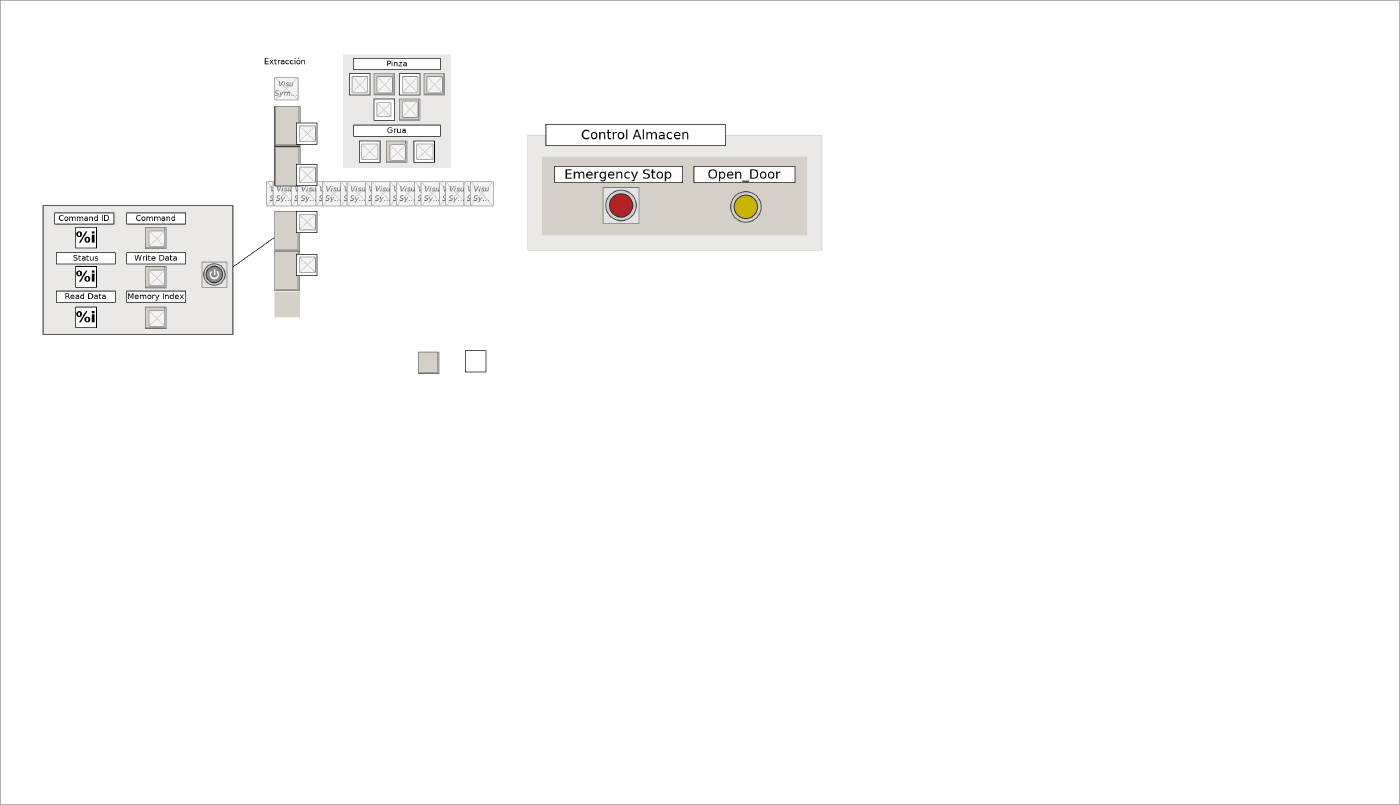
VISUALIZATION Almacen_Manual  // 1930x1110
    Rectangle (369,356 55x35), angle 90
    Group (367,250 330x48)
        Group (0,0 126x48)
            Group (0,0 92x48)
                Group (0,0 58x48)
                    Rectangle (8,5 24x23)
                    Image (0,0 32x34), image: VisuSymbols.Symbols.ArrowForward
                    Image (9,0 32x34), angle 90, image: VisuSymbols.Symbols.ArrowDown
                Group (34,0 58x48)
                    Rectangle (8,5 24x23)
                    Image (0,0 32x34), image: VisuSymbols.Symbols.ArrowForward
                    Image (9,0 32x34), angle 90, image: VisuSymbols.Symbols.ArrowDown
            Group (68,0 58x48)
                Rectangle (8,5 24x23)
                Image (0,0 32x34), image: VisuSymbols.Symbols.ArrowForward
                Image (9,0 32x34), angle 90, image: VisuSymbols.Symbols.ArrowDown
        Group (102,0 126x48)
            Group (0,0 92x48)
                Group (0,0 58x48)
                    Rectangle (8,5 24x23)
                    Image (0,0 32x34), image: VisuSymbols.Symbols.ArrowForward
                    Image (9,0 32x34), angle 90, image: VisuSymbols.Symbols.ArrowDown
                Group (34,0 58x48)
                    Rectangle (8,5 24x23)
                    Image (0,0 32x34), image: VisuSymbols.Symbols.ArrowForward
                    Image (9,0 32x34), angle 90, image: VisuSymbols.Symbols.ArrowDown
            Group (68,0 58x48)
                Rectangle (8,5 24x23)
                Image (0,0 32x34), image: VisuSymbols.Symbols.ArrowForward
                Image (9,0 32x34), angle 90, image: VisuSymbols.Symbols.ArrowDown
        Group (204,0 126x48)
            Group (0,0 92x48)
                Group (0,0 58x48)
                    Rectangle (8,5 24x23)
                    Image (0,0 32x34), image: VisuSymbols.Symbols.ArrowForward
                    Image (9,0 32x34), angle 90, image: VisuSymbols.Symbols.ArrowDown
                Group (34,0 58x48)
                    Rectangle (8,5 24x23)
                    Image (0,0 32x34), image: VisuSymbols.Symbols.ArrowForward
                    Image (9,0 32x34), angle 90, image: VisuSymbols.Symbols.ArrowDown
            Group (68,0 58x48)
                Rectangle (8,5 24x23)
                Image (0,0 32x34), image: VisuSymbols.Symbols.ArrowForward
                Image (9,0 32x34), angle 90, image: VisuSymbols.Symbols.ArrowDown
    InvisibleInput (355,103 77x35)
    Image (378,106 33x32), image: VisuSymbols.Symbols.ForwardStandard
    Rectangle (347,76 92x18), "Extracción"
    Rectangle (379,402 35x35), angle 90
    Rectangle (369,301 55x35), angle 90
    Rectangle (369,211 55x35), angle 90
    Rectangle (369,156 55x35), angle 90
    InvisibleInput (1163,198 18x136)
    Line (377,328) (318,370)
    InvisibleInput (262,497 18x41)
    Rectangle (1771,538 159x406), angle 90
    Rectangle (752,171 248x30), "Control Almacen"
    Rectangle (1780,528 108x365), angle 90
    PushSwitch (831,258 50x50), variable: GVL.Emergency_Stop_9, behaviour: TOGGLE, style: Switch-PushSwitch-Red
    Rectangle (764,229 177x23), "Emergency Stop"
    Lamp1 (1003,260 50x50), variable: NOT GVL.Safety_Door_13 OR NOT GVL.Safety_Door_14 OR NOT GVL.Safety_Door_15, style: Lamp-Lamp1-Yellow
    Rectangle (956,229 140x23), "Open_Door"
    Rectangle (1198,848 178x262), angle 90
    Rectangle (104,313 29x29), "%i", text variable: GVL.RFID_Reader_1_Command_ID
        p4168582468: GVL.RFID_Reader_1_Command_ID
    Rectangle (75,293 82x16), "Command ID"
    Rectangle (77,348 82x16), "Status"
    Rectangle (77,401 82x16), "Read Data"
    Rectangle (104,367 29x29), "%i", text variable: GVL.RFID_Reader_1_Status
        p4168582468: GVL.RFID_Reader_1_Status
    Rectangle (104,423 29x29), "%i", text variable: GVL.RFID_Reader_1_Read_Data
        p4168582468: GVL.RFID_Reader_1_Read_Data
    PowerSwitch (278,361 35x35), variable: GVL.RFID_Reader_1_Ejecute_Comm, behaviour: TOGGLE, style: Switch-PowerSwitch-Gray
    Button (378,346 35x55), colour toggle: GVL.Roller_Conveyor_2m_8, pressed state: GVL.Roller_Conveyor_2m_8
        OnMouseClick: toggle GVL.Roller_Conveyor_2m_8
    Button (378,291 35x55), colour toggle: GVL.Loading_Conveyor_1, pressed state: GVL.Loading_Conveyor_1
        OnMouseClick: toggle GVL.Loading_Conveyor_1
    Group (408,291 29x30), colour toggle: GVL.Retroreflective_Sensor_1
        RoundedRectangle (0,0 29x30), colour toggle: GVL.Diffuse_Sensor_4
        Image (4,4 23x22), image: VisuSymbols.Symbols.RSS1
    Group (408,350 29x30), colour toggle: GVL.Diffuse_Sensor_43
        RoundedRectangle (0,0 29x30), colour toggle: GVL.Diffuse_Sensor_4
        Image (4,4 23x22), image: VisuSymbols.Symbols.RSS1
    Button (379,202 35x55), colour toggle: GVL.Loading_Conveyor_2, pressed state: GVL.Loading_Conveyor_2
        OnMouseClick: toggle GVL.Loading_Conveyor_2
    Button (379,146 35x55), colour toggle: GVL.Roller_Conveyor_2m_9, pressed state: GVL.Roller_Conveyor_2m_9
        OnMouseClick: toggle GVL.Roller_Conveyor_2m_9
    Group (408,226 29x30), colour toggle: GVL.Retroreflective_Sensor_2
        RoundedRectangle (0,0 29x30), colour toggle: GVL.Diffuse_Sensor_4
        Image (4,4 23x22), image: VisuSymbols.Symbols.RSS1
    Group (408,169 29x30), colour toggle: GVL.Diffuse_Sensor_44
        RoundedRectangle (0,0 29x30), colour toggle: GVL.Diffuse_Sensor_4
        Image (4,4 23x22), image: VisuSymbols.Symbols.RSS1
    Rectangle (1505,647 156x148), angle 90
    Rectangle (487,80 120x16), "Pinza"
    Group (495,194 29x30), colour toggle: GVL.Stacker_Crane_1_Moving_X
        RoundedRectangle (0,0 29x30), colour toggle: GVL.Diffuse_Sensor_4
        Image (3,4 23x22), image: VisuSymbols.Symbols.DoubleArrow3
    Group (570,194 29x30), colour toggle: GVL.Stacker_Crane_1_Moving_Z
        RoundedRectangle (0,0 29x30), colour toggle: GVL.Diffuse_Sensor_4
        Image (4,4 23x22), image: VisuSymbols.Symbols.DoubleArrow4
    Rectangle (487,172 120x16), "Grua"
    Group (550,136 29x30), colour toggle: GVL.Stacker_Crane_1_Lift
        OnMouseClick: toggle GVL.Stacker_Crane_1_Lift
        Button (0,0 29x30), colour toggle: GVL.Stacker_Crane_1_Lift
        Image (4,3 22x23), image: VisuSymbols.Symbols.ArrowBoldUp
    Button (515,101 29x30)
    Image (519,105 22x23), colour toggle: GVL.Stacker_Crane_1_Left, image: VisuSymbols.Symbols.ArrowBoldLeft
        OnMouseClick: toggle GVL.Stacker_Crane_1_Left
    Group (481,101 29x30), colour toggle: GVL.Stacker_Crane_1_Left_Limit
        RoundedRectangle (0,0 29x30), colour toggle: GVL.Diffuse_Sensor_4
        Image (4,4 22x23), image: VisuSymbols.Symbols.ArrowBoldLeft
    Group (584,101 29x30), colour toggle: GVL.Stacker_Crane_1_Right
        OnMouseClick: toggle GVL.Stacker_Crane_1_Right
        Button (0,0 29x30)
        Image (4,4 22x23), image: VisuSymbols.Symbols.ArrowBoldRight
    Group (550,101 29x30), colour toggle: GVL.Stacker_Crane_1_Right_Limit
        RoundedRectangle (0,0 29x30), colour toggle: GVL.Diffuse_Sensor_4
        Image (4,4 22x23), image: VisuSymbols.Symbols.ArrowBoldRight
    Group (515,136 29x30), colour toggle: NOT GVL.Stacker_Crane_1_Middle_Limit
        RoundedRectangle (0,0 29x30), colour toggle: GVL.Diffuse_Sensor_4
        Image (4,5 20x20), angle 135, image: VisuSymbols.Symbols.DoubleArrow1
    Rectangle (174,293 82x16), "Command"
    Rectangle (174,348 82x16), "Write Data"
    Rectangle (174,401 82x16), "Memory Index"
    Group (200,313 29x30)
        OnMouseClick: write GVL.RFID_Reader_4_Command_ID via VisuDialogs.Numpad, min 0, max 100, format %i
        Button (0,0 29x30), text variable: GVL.RFID_Reader_1_Command
            OnMouseClick: write GVL.RFID_Reader_4_Command_ID via VisuDialogs.Numpad, min 0, max 100, format %i
        Image (5,5 22x22), image: VisuSymbols.Symbols.Edit
    Group (200,367 29x30)
        OnMouseClick: write GVL.RFID_Reader_4_Write_Data via VisuDialogs.Numpad, min 0, max 100, format %i
        Button (0,0 29x30), text variable: GVL.RFID_Reader_1_Command
            OnMouseClick: write GVL.RFID_Reader_4_Command_ID via VisuDialogs.Numpad, min 0, max 100, format %i
        Image (5,5 22x22), image: VisuSymbols.Symbols.Edit
    Group (200,423 29x30)
        OnMouseClick: write GVL.RFID_Reader_4_Memory_Index via VisuDialogs.Numpad, min 0, max 100, format %i
        Button (0,0 29x30), text variable: GVL.RFID_Reader_1_Command
            OnMouseClick: write GVL.RFID_Reader_4_Command_ID via VisuDialogs.Numpad, min 0, max 100, format %i
        Image (5,5 22x22), image: VisuSymbols.Symbols.Edit
    Group (532,194 29x30)
        OnMouseClick: write GVL.Stacker_Crane_1_Target_Position via VisuDialogs.Numpad, min 0, max 53, format %i
        Button (0,0 29x30), text variable: GVL.RFID_Reader_1_Command
            OnMouseClick: write GVL.RFID_Reader_4_Command_ID via VisuDialogs.Numpad, min 0, max 100, format %i
        Image (5,5 22x22), image: VisuSymbols.Symbols.Edit
    Button (576,485 29x30), text variable: GVL.RFID_Reader_1_Command
        OnMouseClick: write GVL.RFID_Reader_4_Command_ID via VisuDialogs.Numpad, min 0, max 100, format %i
    RoundedRectangle (641,483 29x30), colour toggle: GVL.Diffuse_Sensor_4
END_VISUALIZATION

(* stored: Version 1.1.0.1, ProductVersion 3.1.4024.12
   Visu Almacen_Manual: Id {fb3c63bd-4b24-470a-9c55-a218dbeb1702} *)
